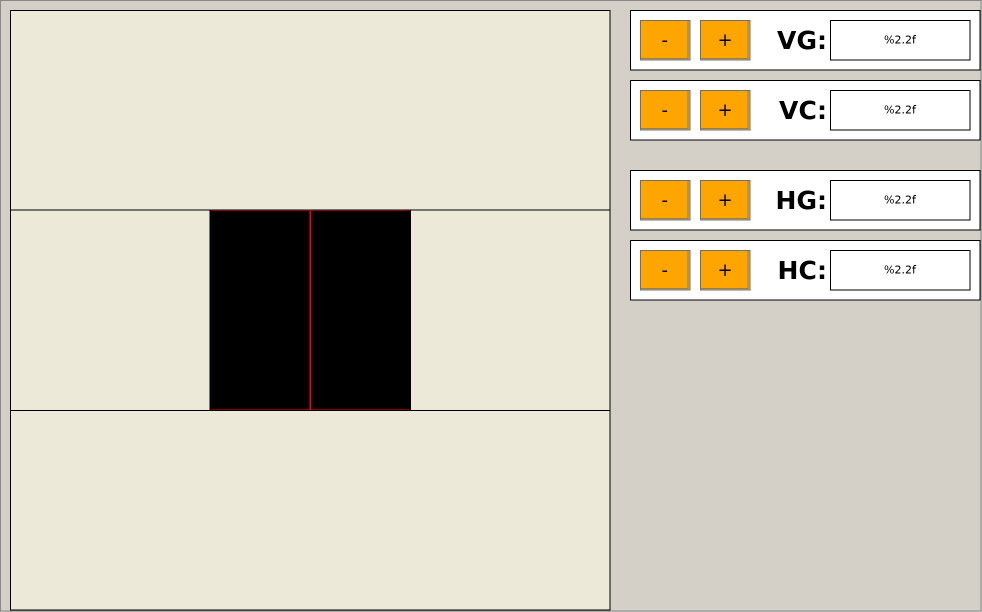
VISUALIZATION SlitSet  // 982x612
    Rectangle (630,10 350x60)
    Rectangle (210,210 200x200)
    Rectangle (210,160 200x150)
        p2738717112: -GVL.axes[1].Axis.NcToPlc.ActPos
    Rectangle (210,310 200x150)
        p2738717112: -GVL.axes[2].Axis.NcToPlc.ActPos
    Rectangle (310,210 150x200)
        p3560616238: GVL.axes[3].Axis.NcToPlc.ActPos
    Rectangle (160,210 150x200)
        p3560616238: GVL.axes[4].Axis.NcToPlc.ActPos
    Rectangle (410,160 200x300)
    Rectangle (10,160 200x300)
    Rectangle (10,10 600x200)
    Rectangle (10,410 600x200)
    Textfield (830,20 140x40), "%2.2f", text variable: GVL.axes[5].Axis.NcToPlc.ActPos
    Button (700,20 50x40), "+"
        tap GVL.axes[5].bJogForward
        OnMouseClick: execute { GVL.axes[5].eCommand:=eMcCommand.Jog; }
    Button (640,20 50x40), "-"
        tap GVL.axes[5].bJogBackward
        OnMouseClick: execute { GVL.axes[5].eCommand:=eMcCommand.Jog; }
    Textfield (760,20 70x40), "VG:"
    Rectangle (630,80 350x60)
    Textfield (830,90 140x40), "%2.2f", text variable: GVL.axes[6].Axis.NcToPlc.ActPos
    Button (700,90 50x40), "+"
        tap GVL.axes[6].bJogForward
        OnMouseClick: execute { GVL.axes[6].eCommand:=eMcCommand.Jog; }
    Button (640,90 50x40), "-"
        tap GVL.axes[6].bJogBackward
        OnMouseClick: execute { GVL.axes[6].eCommand:=eMcCommand.Jog; }
    Textfield (760,90 70x40), "VC:"
    Rectangle (630,170 350x60)
    Textfield (830,180 140x40), "%2.2f", text variable: GVL.axes[7].Axis.NcToPlc.ActPos
    Button (700,180 50x40), "+"
        tap GVL.axes[7].bJogForward
        OnMouseClick: execute { GVL.axes[7].eCommand:=eMcCommand.Jog; }
    Button (640,180 50x40), "-"
        tap GVL.axes[7].bJogBackward
        OnMouseClick: execute { GVL.axes[7].eCommand:=eMcCommand.Jog; }
    Textfield (760,180 70x40), "HG:"
    Rectangle (630,240 350x60)
    Textfield (830,250 140x40), "%2.2f", text variable: GVL.axes[8].Axis.NcToPlc.ActPos
    Button (700,250 50x40), "+"
        tap GVL.axes[8].bJogForward
        OnMouseClick: execute { GVL.axes[8].eCommand:=eMcCommand.Jog; }
    Button (640,250 50x40), "-"
        tap GVL.axes[8].bJogBackward
        OnMouseClick: execute { GVL.axes[8].eCommand:=eMcCommand.Jog; }
    Textfield (760,250 70x40), "HC:"
END_VISUALIZATION

(* stored: Version 1.1.0.1, ProductVersion 3.1.4022.12
   Visu SlitSet: Id {b79c5954-fb2e-4618-aba7-fc55cdc25217} *)
